FUNCTION_BLOCK Control_Observer IMPLEMENTS ITF_Observer
VAR
	SystemSafetyState : INT;
END_VAR

METHOD Update : BOOL
VAR_INPUT
	TwinSAFEState : INT;
END_VAR
SystemSafetyState := TwinSAFEState;
END_METHOD

END_FUNCTION_BLOCK

(* stored: Version 1.1.0.1, ProductVersion 3.1.4024.12
   POU Control_Observer: Id {74fe5921-e5b1-4b65-972d-5c4a51ab573d}, SpecialFunc None
   Method Update: Id {ca0713df-fd81-4182-a262-eff6df3cef60} *)
